// TIA Portal V17 export
// export: Created 2022-03-12T16:05:32.4285237Z, ExportSetting WithDefaults, DisplayName Totally Integrated Automation Portal, DisplayVersion V17, DisplayName TIA Portal Openness, DisplayVersion V17, DisplayName TIA Portal Version Control Interface, DisplayVersion V17, DisplayName STEP 7 Professional, DisplayVersion V17, DisplayName STEP 7 Safety, DisplayVersion V17, DisplayName WinCC Advanced / Unified PC, DisplayVersion V17
VAR_GLOBAL   // PLC tag table "CPG_Constants"
END_VAR
VAR_GLOBAL CONSTANT   // user constants
   CPG_NO_OF_ELEMENTS_EVENT_STATUS_UPPER_LIM : Int := 29;   // Number of Alarms, Warning and PackML Status events used by Event Status UDT (Array size of 0..x)
   CPG_NO_OF_ADMIN_EVENTS_UPPER_LIM : Int := 9;   // Number of Alarms and Warning events found in the PackTags Admin Area - active alarms / warnings. (Array size of 0..x)
   CPG_NO_OF_ADMIN_EVENTS_HISTORY_UPPER_LIM : Int := 9;   // Number of Alarms and Warning events found in the PackTags Admin Area - historical alarms / warnings. (Array size of 0..x)
   CPG_NO_OF_PROD_CONSUMED_COUNT_UPPER_LIM : Int := 0;   // Number of Prod Consumed Counter Array Size (PackTags Admin) (Array size of 0..x)
   CPG_NO_OF_PROD_PROCESSED_COUNT_UPPER_LIM : Int := 0;   // Number of Prod Processed Counter Array Size (PackTags Admin) (Array size of 0..x)
   CPG_NO_OF_PROD_DEFECTIVE_COUNT_UPPER_LIM : Int := 0;   // Number of Prod Defective Counter Array Size (PackTags Admin) (Array size of 0..x)
   CPG_NO_OF_STS_ELEMENTS_EVENT_SUM_UPPER_LIM : Int := 99;   // Number of Alarms, Warning and PackML Status events used by Event Summation UDT (Array size of 0..x)
   CPG_NO_OF_HMI_SORT_EVENTS_UPPER_LIM : Int := 19;   // Number of Alarms and Warning events found for the HMI area - sorted HMI alarms / warnings. (Array size of 0..x)
   CPG_NO_OF_CFG_ALARMS_UPPER_LIM : Int := 39;   // Number of Cfg Alarm event configurations (Array size of 0..x)
   CPG_NO_OF_CFG_WARNINGS_UPPER_LIM : Int := 29;   // Number of Cfg Warning event configurations (Array size of 0..x)
   CPG_NO_OF_CFG_STATUS_UPPER_LIM : Int := 19;   // Number of Cfg Status event configurations (Array size of 0..x)
   CPG_NO_OF_STATUS_PARAMETERS_UPPER_LIM : Int := 0;   // Number of Status Parameters (Array size of 0..x)
   CPG_NO_OF_COMMAND_PARAMETERS_UPPER_LIM : Int := 0;   // Number of Command Parameters (Array size of 0..x)
   CPG_NO_OF_ADMIN_PARAMETERS_UPPER_LIM : Int := 0;   // Number of Admin Parameters (Array size of 0..x)
   CPG_NO_OF_RECIPE_UPPER_LIM : Int := 20;   // Number of Project Recipies (Array size of 0..x)
   CPG_NO_OF_SETPOINT_REAL_UPPER_LIM : Int := 0;   // Number of Setpoints with a REAL type (Array size of 0..x)
   CPG_NO_OF_SETPOINT_DINT_UPPER_LIM : Int := 0;   // Number of Setpoints with a DINT type (Array size of 0..x)
   CPG_NO_OF_SETPOINT_BOOL_UPPER_LIM : Int := 0;   // Number of Setpoints with a BOOL type (Array size of 0..x)
   CPG_NO_OF_SETPOINT_STRING_UPPER_LIM : Int := 0;   // Number of Setpoints with a STRING type (Array size of 0..x)
   CPG_PARTEO_NO_OF_ERRORS_UPPER_LIM : Int := 100;   // Number of Unique Error IDs tracked by PARETO Error Blocks
END_VAR
